# B&R Automation Studio project KeePakST401VersionX (part 5)

#### SafetySample.st
```iecst
(********************************************************************
 * COPYRIGHT -- Bernecker + Rainer
 ********************************************************************
 * Program: SafetySample
 * File: SafetySample.st
 * Author: B&R
 ********************************************************************
 * Implementation of program SafetySample
 ********************************************************************)

PROGRAM _INIT

(*KEEPAK specific hard coded values *)
	remotecmd.Password 			:= 'safety';				(* password *)
	remotecmd.NewPassword	 	:= 'safety';				(* password *)
	appcmd1.Password 			:= 'safety';
	datacmd1.Password 			:= 'safety';
	datacmd2.Password 			:= 'safety';

	visuUsedSLIDRemote			:= 1;
	visuUsedSLIDData			:= 1;

	slxused						:= 1;
	Station						:= 'IF6.ST4';
	visuEnableMachineOptions	:= 1;
	visuEnableModuleFlags		:= 1;

	visuLockSDP					:= 2;

(* command structure for remote control FUB *)
remotecmd.Version := safeVERSION_R107;	(* version *)
//remotecmd.Password := '';				(* password *)

(* command structure for application download *)
appcmd1.Version := safeVERSION_R107;	(* version *)
//appcmd1.Password := '';					(* password *)
appcmd1.ApplicationID := 1;				(* application id *)

(* command structure for machine options download *)
datacmd1.Version := safeVERSION_R107;								(* version *)
//datacmd1.Password := '';											(* password *)
datacmd1.pDeviceListInput := ADR(visuDeviceListInput);				(* device list *)
datacmd1.pMachineOptionsInput := ADR(dataMachineOptionsBitInput);	(* bit machine options *)
datacmd1.pModuleFlagsInput := ADR(dataModuleFlagsInput);			(* module flags *)
datacmd1.pAcknMachineOptions := ADR(dataAcknMachineOptions);		(* acknowledge information *)

(* command structure for extended machine options *)
datacmd2.Version := safeVERSION_R107;					(* version *)
//datacmd2.Password := '';								(* password *)
datacmd2.pIntDataInput := ADR(visuIntInput);			(* INT channels *)
datacmd2.NumberIntInput := 1;							(* number of INT channels *)
datacmd2.pUintDataInput := ADR(visuUintInput);			(* UINT channels *)
datacmd2.NumberUintInput := 1;							(* number of UINT channels *)
datacmd2.pDintDataInput := ADR(visuDintInput);			(* DINT channels *)
datacmd2.NumberDintInput := 1;							(* number of DINT channels *)
datacmd2.pUdintDataInput := ADR(visuUdintInput);		(* UDINT channels *)
datacmd2.NumberUdintInput := 1;							(* number of UDINT channels *)
datacmd2.pAcknMachineOptions := ADR(visuAcknExtData);	(* acknowledge information *)

(* hide elements in visualization *)
FOR xcnt := 0 TO SIZEOF(statusButtonActiv) - 1 DO
	statusButtonActiv[xcnt] := 1;
END_FOR

(* hide elements in visualization *)
statusButtonUnlockApp := 1;
statusButtonUnlockData := 1;
statusAcknInfoData := 1;
statusButtonUnlockExtData := 1;
statusAcknInfoExtData := 1;
statusDialog := 1;

(* set SafeLOGIC ID *)
visuUsedSLIDRemote := 1;
visuUsedSLIDData := 1;

END_PROGRAM

PROGRAM _CYCLIC
	(****************************************************************************************************************************************)
	(****************************************************************************************************************************************)
	(****************************************************************************************************************************************)
	(* show dialog to ackn command *)
	IF (dialogRemoteCmd = 1) THEN
		statusDialog := 0;
		dialogRemoteCmd := 0;
		indexButtonLeft := 0;
		indexButtonRight := 1;
		indexHeaderText := 0;
		IF (remotecmd.Data = safeCMD_SK_FORMAT) THEN
			indexMessageText := 0;
		ELSIF (remotecmd.Data = safeCMD_SK_XCHG) THEN
			indexMessageText := 1;
		ELSIF (remotecmd.Data = safeCMD_1_UDID_ACKN) THEN
			indexMessageText := 2;
		ELSIF (remotecmd.Data = safeCMD_2_UDID_ACKN) THEN
			indexMessageText := 3;
		ELSIF (remotecmd.Data = safeCMD_3_UDID_ACKN) THEN
			indexMessageText := 4;
		ELSIF (remotecmd.Data = safeCMD_4_UDID_ACKN) THEN
			indexMessageText := 5;
		ELSIF (remotecmd.Data =  safeCMD_N_UDID_ACKN) THEN
			indexMessageText := 6;
		ELSIF (remotecmd.Data =  safeCMD_CLEAR_DATA) THEN
			indexMessageText := 7;
		ELSIF (remotecmd.Data = safeCMD_FW_ACKN) THEN
			indexMessageText := 8;
		ELSIF (remotecmd.Data = safeCMD_RESET) THEN
			indexMessageText := 9;
		END_IF
	END_IF

	(* if dialog is ackn execute fub *)
	IF (dialogButtonLeft = 1 AND indexHeaderText = 0) THEN
		executeRemoteCmd := 1;
		dialogButtonLeft := 0;
		statusDialog := 1;
	ELSIF (dialogButtonRight = 1 AND indexHeaderText = 0) THEN
		dialogButtonRight := 0;
		statusDialog := 1;
	END_IF

	(* password must be at least 6 characters long *)
	IF brsstrlen(ADR(remotecmd.NewPassword)) < 6 THEN
		statusSetPassword := 2;
	ELSE
		statusSetPassword := 0;
	END_IF

	safeRemoteControl_0(SafeLOGICID := visuUsedSLIDRemote, Execute := executeRemoteCmd, pCommandData := ADR(remotecmd));
	(* reset execution flag *)
	IF (safeRemoteControl_0.Done = 1 OR safeRemoteControl_0.Error = 1) THEN
		executeRemoteCmd := 0;
	END_IF

	(* variables for visualization *)
	IF (safeRemoteControl_0.SafeLOGICStatus.SafeKEYChanged = 1) THEN
		FOR xcnt := 0 TO SIZEOF(statusButtonActiv) - 1 DO
			statusButtonActiv[xcnt] := 1;
 			statusButtonInactiv[xcnt] := 0;
		END_FOR
		statusButtonActiv[1] := 0;
 		statusButtonInactiv[1] := 1;
	ELSIF (safeRemoteControl_0.SafeLOGICStatus.NumberOfUDIDMismatches = 1 AND safeRemoteControl_0.SafeLOGICStatus.Scanning = 0) THEN
		FOR xcnt := 0 TO SIZEOF(statusButtonActiv) - 1 DO
			statusButtonActiv[xcnt] := 1;
 			statusButtonInactiv[xcnt] := 0;
		END_FOR
		statusButtonActiv[3] := 0;
 		statusButtonInactiv[3] := 1;
	ELSIF (safeRemoteControl_0.SafeLOGICStatus.NumberOfUDIDMismatches = 2 AND safeRemoteControl_0.SafeLOGICStatus.Scanning = 0) THEN
		FOR xcnt := 0 TO SIZEOF(statusButtonActiv) - 1 DO
			statusButtonActiv[xcnt] := 1;
 			statusButtonInactiv[xcnt] := 0;
		END_FOR
		statusButtonActiv[4] := 0;
 		statusButtonInactiv[4] := 1;
	ELSIF (safeRemoteControl_0.SafeLOGICStatus.NumberOfUDIDMismatches = 3 AND safeRemoteControl_0.SafeLOGICStatus.Scanning = 0) THEN
		FOR xcnt := 0 TO SIZEOF(statusButtonActiv) - 1 DO
			statusButtonActiv[xcnt] := 1;
 			statusButtonInactiv[xcnt] := 0;
		END_FOR
		statusButtonActiv[5] := 0;
 		statusButtonInactiv[5] := 1;
	ELSIF (safeRemoteControl_0.SafeLOGICStatus.NumberOfUDIDMismatches = 4 AND safeRemoteControl_0.SafeLOGICStatus.Scanning = 0) THEN
		FOR xcnt := 0 TO SIZEOF(statusButtonActiv) - 1 DO
			statusButtonActiv[xcnt] := 1;
 			statusButtonInactiv[xcnt] := 0;
		END_FOR
		statusButtonActiv[6] := 0;
 		statusButtonInactiv[6] := 1;
	ELSIF (safeRemoteControl_0.SafeLOGICStatus.NumberOfUDIDMismatches > 4 AND safeRemoteControl_0.SafeLOGICStatus.Scanning = 0) THEN
		FOR xcnt := 0 TO SIZEOF(statusButtonActiv) - 1 DO
			statusButtonActiv[xcnt] := 1;
 			statusButtonInactiv[xcnt] := 0;
		END_FOR
		statusButtonActiv[7] := 0;
 		statusButtonInactiv[7] := 1;
	ELSIF (safeRemoteControl_0.SafeLOGICStatus.NumberOfDifferentFirmware <> 0 AND safeRemoteControl_0.SafeLOGICStatus.Scanning = 0) THEN
		FOR xcnt := 0 TO SIZEOF(statusButtonActiv) - 1 DO
			statusButtonActiv[xcnt] := 1;
 			statusButtonInactiv[xcnt] := 0;
		END_FOR
		statusButtonActiv[11] := 0;
 		statusButtonInactiv[11] := 1;
	ELSE
		FOR xcnt := 0 TO SIZEOF(statusButtonActiv) - 1 DO
			statusButtonActiv[xcnt] := 1;
 			statusButtonInactiv[xcnt] := 0;
		END_FOR
	END_IF
	(* status text - MXCHG *)
	IF (safeRemoteControl_0.SafeLOGICStatus.LedTestActive = 1) THEN
		indexMxchgLed := 40;
	ELSIF (safeRemoteControl_0.SafeLOGICStatus.Scanning = 1) THEN
		indexMxchgLed := 30;
	ELSIF (safeRemoteControl_0.SafeLOGICStatus.NumberOfUDIDMismatches = 1) THEN
		indexMxchgLed := 1;
	ELSIF (safeRemoteControl_0.SafeLOGICStatus.NumberOfUDIDMismatches = 2) THEN
		indexMxchgLed := 2;
	ELSIF (safeRemoteControl_0.SafeLOGICStatus.NumberOfUDIDMismatches = 3) THEN
		indexMxchgLed := 3;
	ELSIF (safeRemoteControl_0.SafeLOGICStatus.NumberOfUDIDMismatches = 4) THEN
		indexMxchgLed := 4;
	ELSIF (safeRemoteControl_0.SafeLOGICStatus.NumberOfUDIDMismatches > 4) THEN
		indexMxchgLed := 5;
	ELSIF (safeRemoteControl_0.SafeLOGICStatus.NumberOfMissingModules <> 0) THEN
		indexMxchgLed := 20;
	ELSIF (safeRemoteControl_0.SafeLOGICStatus.NumberOfUDIDMismatches = 0) THEN
		indexMxchgLed := 10;
	END_IF
	(* status text - FW-ACKN *)
	IF (safeRemoteControl_0.SafeLOGICStatus.SafeKEYChanged = 0 AND safeRemoteControl_0.SafeLOGICStatus.NumberOfDifferentFirmware = 0) THEN
		indexFwAcknLed := 10;
	ELSIF (safeRemoteControl_0.SafeLOGICStatus.SafeKEYChanged = 1) THEN
		indexFwAcknLed := 1;
	ELSIF (safeRemoteControl_0.SafeLOGICStatus.NumberOfDifferentFirmware <> 0) THEN
		indexFwAcknLed := 2;
	END_IF
	(* status text - FAIL *)
	IF (safeRemoteControl_0.SafeLOGICStatus.FailSafe <> 16#55) THEN
		indexFAILLed := 2;
	ELSIF (safeRemoteControl_0.SafeLOGICStatus.openSAFETYstate = 0) THEN
		indexFAILLed := 0;
	ELSIF (safeRemoteControl_0.SafeLOGICStatus.openSAFETYstate = 1) THEN
		indexFAILLed := 1;
	END_IF
	(* status text - R/E *)
	indexRELed := safeRemoteControl_0.SafeLOGICStatus.SafeOSState;

	(****************************************************************************************************************************************)
	(****************************************************************************************************************************************)
	(****************************************************************************************************************************************)
	(* show dialog to ackn command *)
	IF (dialogApplication = 1) THEN
		statusDialog := 0;
		dialogApplication := 0;
		indexButtonLeft := 0;
		indexButtonRight := 1;
		indexHeaderText := 1;
		indexMessageText := 10;
	END_IF

	(* if dialog is ackn unlock application *)
	IF (dialogButtonLeft = 1 AND indexHeaderText = 1) THEN
		appcmd1.Unlock := 1;
		dialogButtonLeft := 0;
		statusDialog := 1;
	ELSIF (dialogButtonRight = 1 AND indexHeaderText = 1) THEN
		appcmd1.Unlock := 2;
		dialogButtonRight := 0;
		statusDialog := 1;
	END_IF

	(* convert application CRC to HEX string *)
	itoahex(safeDownloadApplication_0.ApplicationCRC, ADR(visuApplicationCRC));

	safeDownloadApplication_0(SafeLOGICID := appcmd1.ApplicationID, Execute := executeapp1, pCommandData := ADR(appcmd1));

	(* show unlock button *)
	IF (safeDownloadApplication_0.UnlockRequired = 1) THEN
		statusButtonUnlockApp := 0;
	ELSE
		appcmd1.Unlock := 0;
		statusButtonUnlockApp := 1;
	END_IF

	(****************************************************************************************************************************************)
	(****************************************************************************************************************************************)
	(****************************************************************************************************************************************)
	(* disable machine options *)
	IF (visuEnableMachineOptions = FALSE) THEN
		datacmd1.pMachineOptionsInput := 0;
	ELSE
		datacmd1.pMachineOptionsInput := ADR(dataMachineOptionsBitInput);
	END_IF

	(* disable module flags *)
	IF (visuEnableModuleFlags = FALSE) THEN
		datacmd1.pModuleFlagsInput := 0;
	ELSE
		datacmd1.pModuleFlagsInput := ADR(dataModuleFlagsInput);
	END_IF

	(* Machine Option Bit #000 *)
	IF (visuMachineOptionsBitInput[0] = 1) THEN
		dataMachineOptionsBitInput.BitData[0].0 := 1;
	ELSE
		dataMachineOptionsBitInput.BitData[0].0 := 0;
	END_IF
	(* Machine Option Bit #001 *)
	IF (visuMachineOptionsBitInput[1] = 1) THEN
		dataMachineOptionsBitInput.BitData[0].1 := 1;
	ELSE
		dataMachineOptionsBitInput.BitData[0].1 := 0;
	END_IF
	(* Machine Option Bit #002 *)
	IF (visuMachineOptionsBitInput[2] = 1) THEN
		dataMachineOptionsBitInput.BitData[0].2 := 1;
	ELSE
		dataMachineOptionsBitInput.BitData[0].2 := 0;
	END_IF
	(* Optional Flag Module #1 *)
	IF (visuModuleFlagsOptionalInput[1] = 1) THEN
		dataModuleFlagsInput.Optional[0].1 := 1;
	ELSE
		dataModuleFlagsInput.Optional[0].1 := 0;
	END_IF
	(* Optional Flag Module #2 *)
	IF (visuModuleFlagsOptionalInput[2] = 1) THEN
		dataModuleFlagsInput.Optional[0].2 := 1;
	ELSE
		dataModuleFlagsInput.Optional[0].2 := 0;
	END_IF
	(* Startup Flag Module #1 *)
	IF (visuModuleFlagsStartupInput[1] = 1) THEN
		dataModuleFlagsInput.Startup[0].1 := 1;
	ELSE
		dataModuleFlagsInput.Startup[0].1 := 0;
	END_IF
	(* Startup Flag Module #2 *)
	IF (visuModuleFlagsStartupInput[2] = 1) THEN
		dataModuleFlagsInput.Startup[0].2 := 1;
	ELSE
		dataModuleFlagsInput.Startup[0].2 := 0;
	END_IF
	(* Not_Present Flag Module #1 *)
	IF (visuModuleFlagsNotPresentInput[1] = 1) THEN
		dataModuleFlagsInput.NotPresent[0].1 := 1;
	ELSE
		dataModuleFlagsInput.NotPresent[0].1 := 0;
	END_IF
	(* Not_Present Flag Module #2 *)
	IF (visuModuleFlagsNotPresentInput[2] = 1) THEN
		dataModuleFlagsInput.NotPresent[0].2 := 1;
	ELSE
		dataModuleFlagsInput.NotPresent[0].2 := 0;
	END_IF

	(* Ackn Machine Option Bit #000 *)
	IF (visuAcknMachineOptions[0] = 1) THEN
		dataAcknMachineOptions.AcknBitOptions[0].0 := 1;
	ELSE
		dataAcknMachineOptions.AcknBitOptions[0].0 := 0;
	END_IF
	(* Ackn Machine Option Bit #001 *)
	IF (visuAcknMachineOptions[1] = 1) THEN
		dataAcknMachineOptions.AcknBitOptions[0].1 := 1;
	ELSE
		dataAcknMachineOptions.AcknBitOptions[0].1 := 0;
	END_IF
	(* Ackn Machine Option Bit #002 *)
	IF (visuAcknMachineOptions[2] = 1) THEN
		dataAcknMachineOptions.AcknBitOptions[0].2 := 1;
	ELSE
		dataAcknMachineOptions.AcknBitOptions[0].2 := 0;
	END_IF

	(* show dialog to ackn command *)
	IF (dialogData = 1) THEN
		statusDialog := 0;
		dialogData := 0;
		indexButtonLeft := 0;
		indexButtonRight := 1;
		indexHeaderText := 2;
		indexMessageText := 11;
	END_IF

	(* if dialog is ackn unlock data *)
	IF (dialogButtonLeft = 1 AND indexHeaderText = 2) THEN
		datacmd1.Unlock := 1;
		dialogButtonLeft := 0;
		statusDialog := 1;
	ELSIF (dialogButtonRight = 1 AND indexHeaderText = 2) THEN
		datacmd1.Unlock := 2;
		dialogButtonRight := 0;
		statusDialog := 1;
	END_IF

	safeDownloadData_0(SafeLOGICID := visuUsedSLIDData, Execute := executedata1, Type:= safeDATA_TYPE_MAOP, pCommandData := ADR(datacmd1));

	(* data compare failed *)
	IF (safeDownloadData_0.StatusID = safeERR_DL_COMPARE_FAILED) THEN
		indexCompareTextData := 2;
	ELSE
		indexCompareTextData := 0;
	END_IF

	IF (safeDownloadData_0.UnlockRequired = 1) THEN
		(* data compare successful *)
		indexCompareTextData := 1;
		IF (datacmd1.pDeviceListOutput <> 0 AND datacmd1.NumberDevicesOutput <> 0) THEN
			pDeviceListOut ACCESS datacmd1.pDeviceListOutput;

			(* device #1 *)
			visuDeviceListOutput[0].SADR := pDeviceListOut[0].SADR;
			brsmemcpy(ADR(visuDeviceListOutput[0].UDID_High), ADR(pDeviceListOut[0].UDID[0]), 2);
			(* swap UDID *)
			visuDeviceListOutput[0].UDID_High := swapUINT(visuDeviceListOutput[0].UDID_High);
			brsmemcpy(ADR(visuDeviceListOutput[0].UDID_Low), ADR(pDeviceListOut[0].UDID[2]), 4);
			(* swap UDID *)
			visuDeviceListOutput[0].UDID_Low := swapUDINT(visuDeviceListOutput[0].UDID_Low);
			(* device #2 *)
			visuDeviceListOutput[1].SADR := pDeviceListOut[1].SADR;
			brsmemcpy(ADR(visuDeviceListOutput[1].UDID_High), ADR(pDeviceListOut[1].UDID[0]), 2);
			(* swap UDID *)
			visuDeviceListOutput[1].UDID_High := swapUINT(visuDeviceListOutput[1].UDID_High);
			brsmemcpy(ADR(visuDeviceListOutput[1].UDID_Low), ADR(pDeviceListOut[1].UDID[2]), 4);
			(* swap UDID *)
			visuDeviceListOutput[1].UDID_Low := swapUDINT(visuDeviceListOutput[1].UDID_Low);
		END_IF

		IF (datacmd1.pMachineOptionsOutput <> 0) THEN
			pMachineOptionsBitOut ACCESS datacmd1.pMachineOptionsOutput;

			(* Machine Option Bit #000 *)
			IF (pMachineOptionsBitOut.BitData[0].0 = 1) THEN
				visuMachineOptionsBitOutput[0] := 1;
			END_IF
			(* Machine Option Bit #001 *)
			IF (pMachineOptionsBitOut.BitData[0].1 = 1) THEN
				visuMachineOptionsBitOutput[1] := 1;
			END_IF
			(* Machine Option Bit #002 *)
			IF (pMachineOptionsBitOut.BitData[0].2 = 1) THEN
				visuMachineOptionsBitOutput[2] := 1;
			END_IF
		END_IF

		IF (datacmd1.pModuleFlagsOutput <> 0) THEN
			pModuleFlagsOut ACCESS datacmd1.pModuleFlagsOutput;

			(* Optional Flag Module #1 *)
			IF (pModuleFlagsOut.Optional[0].1 = 1) THEN
				visuModuleFlagsOptionalOutput[1] := 1;
			END_IF
			(* Optional Flag Module #2 *)
			IF (pModuleFlagsOut.Optional[0].2 = 1) THEN
				visuModuleFlagsOptionalOutput[2] := 1;
			END_IF
			(* Startup Flag Module #1 *)
			IF (pModuleFlagsOut.Startup[0].1 = 1) THEN
				visuModuleFlagsStartupOutput[1] := 1;
			END_IF
			(* Startup Flag Module #2 *)
			IF (pModuleFlagsOut.Startup[0].2 = 1) THEN
				visuModuleFlagsStartupOutput[2] := 1;
			END_IF
			(* Not_Present Flag Module #1 *)
			IF (pModuleFlagsOut.NotPresent[0].1 = 1) THEN
				visuModuleFlagsNotPresentOutput[1] := 1;
			END_IF
			(* Not_Present Flag Module #2 *)
			IF (pModuleFlagsOut.NotPresent[0].2 = 1) THEN
				visuModuleFlagsNotPresentOutput[2] := 1;
			END_IF
		END_IF
		(* show ackn box *)
		statusAcknInfoData := 0;
		(* show unlock button unlocked if one ACK is set *)
		IF (visuAcknMachineOptions[0] = 1 OR visuAcknMachineOptions[1] = 1 OR visuAcknMachineOptions[2] = 1) THEN
			statusButtonUnlockData := 0;
		END_IF
	ELSIF (safeDownloadData_0.Done = 1 OR safeDownloadData_0.Error = 1) THEN
		(* reset visualization elements *)
		brsmemset(ADR(visuDeviceListOutput), 0, SIZEOF(visuDeviceListOutput));
		brsmemset(ADR(visuMachineOptionsBitOutput), 0, SIZEOF(visuMachineOptionsBitOutput));
		brsmemset(ADR(visuModuleFlagsOptionalOutput), 0, SIZEOF(visuModuleFlagsOptionalOutput));
		brsmemset(ADR(visuModuleFlagsStartupOutput), 0, SIZEOF(visuModuleFlagsStartupOutput));
		brsmemset(ADR(visuModuleFlagsNotPresentOutput), 0, SIZEOF(visuModuleFlagsNotPresentOutput));
		(* hide ackn box *)
		statusAcknInfoData := 1;
		(* hide unlock button *)
		datacmd1.Unlock := 0;
		statusButtonUnlockData := 1;
		(* reset ackn flags *)
		visuAcknMachineOptions[0] := 0;
		visuAcknMachineOptions[1] := 0;
		visuAcknMachineOptions[2] := 0;
	ELSE
		(* hide ackn box *)
		statusAcknInfoData := 1;
		(* hide unlock button *)
		datacmd1.Unlock := 0;
		statusButtonUnlockData := 1;
	END_IF

	(****************************************************************************************************************************************)
	(****************************************************************************************************************************************)
	(****************************************************************************************************************************************)
	(* Enable for INT set *)
	IF (visuEnableINTOptions <> 0) THEN
		datacmd2.pIntDataInput := ADR(visuIntInput);
		datacmd2.NumberIntInput := 1;
	ELSE
		datacmd2.pIntDataInput := 0;
		datacmd2.NumberIntInput := 0;
	END_IF
	(* Enable for UINT set *)
	IF (visuEnableUINTOptions <> 0) THEN
		datacmd2.pUintDataInput := ADR(visuUintInput);
		datacmd2.NumberUintInput := 1;
	ELSE
		datacmd2.pUintDataInput := 0;
		datacmd2.NumberUintInput := 0;
	END_IF
	(* Enable for DINT set *)
	IF (visuEnableDINTOptions <> 0) THEN
		datacmd2.pDintDataInput := ADR(visuDintInput);
		datacmd2.NumberDintInput := 1;
	ELSE
		datacmd2.pDintDataInput := 0;
		datacmd2.NumberDintInput := 0;
	END_IF
	(* Enable for UDINT set *)
	IF (visuEnableUDINTOptions <> 0) THEN
		datacmd2.pUdintDataInput := ADR(visuUdintInput);
		datacmd2.NumberUdintInput := 1;
	ELSE
		datacmd2.pUdintDataInput := 0;
		datacmd2.NumberUdintInput := 0;
	END_IF

	(* show dialog to ackn command *)
	IF (dialogExtData = 1) THEN
		statusDialog := 0;
		dialogExtData := 0;
		indexButtonLeft := 0;
		indexButtonRight := 1;
		indexHeaderText := 3;
		indexMessageText := 11;
	END_IF

	(* if dialog is ackn unlock data *)
	IF (dialogButtonLeft = 1 AND indexHeaderText = 3) THEN
		datacmd2.Unlock := 1;
		dialogButtonLeft := 0;
		statusDialog := 1;
	ELSIF (dialogButtonRight = 1 AND indexHeaderText = 3) THEN
		datacmd2.Unlock := 2;
		dialogButtonRight := 0;
		statusDialog := 1;
	END_IF

	safeDownloadData_1(SafeLOGICID := visuUsedSLIDData, Execute := executedata2, Type:= safeDATA_TYPE_EXTMAOP, pCommandData := ADR(datacmd2));

	(* data compare failed *)
	IF (safeDownloadData_1.StatusID = safeERR_DL_COMPARE_FAILED) THEN
		indexCompareTextExtData := 2;
	ELSE
		indexCompareTextExtData := 0;
	END_IF

	IF (safeDownloadData_1.UnlockRequired = 1) THEN
		(* data compare successful *)
		indexCompareTextExtData := 1;

		(* INT channels *)
		IF (datacmd2.pIntDataOutput <> 0 AND datacmd2.NumberIntOutput <> 0) THEN
			brsmemcpy(ADR(visuIntOutput), datacmd2.pIntDataOutput, SIZEOF(visuIntOutput));
		END_IF
		(* UINT channels *)
		IF (datacmd2.pUintDataOutput <> 0 AND datacmd2.NumberUintOutput <> 0) THEN
			brsmemcpy(ADR(visuUintOutput), datacmd2.pUintDataOutput, SIZEOF(visuUintOutput));
		END_IF
		(* DINT channels *)
		IF (datacmd2.pDintDataOutput <> 0 AND datacmd2.NumberDintOutput <> 0) THEN
			brsmemcpy(ADR(visuDintOutput), datacmd2.pDintDataOutput, SIZEOF(visuDintOutput));
		END_IF
		(* UDINT channels *)
		IF (datacmd2.pUdintDataOutput <> 0 AND datacmd2.NumberUdintOutput <> 0) THEN
			brsmemcpy(ADR(visuUdintOutput), datacmd2.pUdintDataOutput, SIZEOF(visuUdintOutput));
		END_IF
		(* show ackn box *)
		statusAcknInfoExtData := 0;
		(* show unlock button if one ACK is set *)
		IF (visuAcknExtData.AcknIntOptions[0] = 1 OR visuAcknExtData.AcknUintOptions[0] = 1 OR visuAcknExtData.AcknDintOptions[0] = 1 OR visuAcknExtData.AcknUdintOptions[0] = 1) THEN
			statusButtonUnlockExtData := 0;
		END_IF
	ELSIF (safeDownloadData_1.Done = 1 OR safeDownloadData_1.Error = 1) THEN
		(* reset visualization elements *)
		brsmemset(ADR(visuIntOutput), 0, SIZEOF(visuIntOutput));
		brsmemset(ADR(visuUintOutput), 0, SIZEOF(visuUintOutput));
		brsmemset(ADR(visuDintOutput), 0, SIZEOF(visuDintOutput));
		brsmemset(ADR(visuUdintOutput), 0, SIZEOF(visuUdintOutput));
		(* hide ackn box *)
		statusAcknInfoExtData := 1;
		(* hide unlock button *)
		datacmd2.Unlock := 0;
		statusButtonUnlockExtData := 1;
		(* reset ackn flags *)
		visuAcknExtData.AcknIntOptions[0] := 0;
		visuAcknExtData.AcknUintOptions[0] := 0;
		visuAcknExtData.AcknDintOptions[0] := 0;
		visuAcknExtData.AcknUdintOptions[0] := 0;
	ELSE
		(* hide ackn box *)
		statusAcknInfoExtData := 1;
		(* hide unlock button *)
		datacmd2.Unlock := 0;
		statusButtonUnlockExtData := 1;
	END_IF

	(****************************************************************************************************************************************)
	(****************************************************************************************************************************************)
	(****************************************************************************************************************************************)
	(* read UDID from SafeLOGIC-X *)
	IF slxused = 1 THEN
		readUDIDlowSLX(enable := 1, pDeviceName := ADR(Station), pChannelName := ADR('UDID_low'));

		IF readUDIDlowSLX.status = 0 THEN
			UDID_Low := readUDIDlowSLX.value;
		ELSIF readUDIDlowSLX.status <> 65535 THEN
			UDID_Low := 0;
		END_IF

		readUDIDhighSLX(enable := 1, pDeviceName := ADR(Station), pChannelName := ADR('UDID_high'));

		IF readUDIDhighSLX.status = 0 THEN
			UDID_High := UDINT_TO_UINT(readUDIDhighSLX.value);
		ELSIF readUDIDhighSLX.status <> 65535 THEN
			UDID_High := 0;
		END_IF

		(* hide / show visualization elements *)
		stautsSLXInformation := 0;
		statusSLInformation := 1;
	(* read UDID form SafeLOGIC *)
	ELSE
		readUDIDlowSL(enable := 1, pDevice := ADR(Interface), node := Node, index := 16#2000, subindex := 6, pData := ADR(UDID_Low), datalen := SIZEOF(UDID_Low));

		IF readUDIDlowSL.status <> 0 AND readUDIDlowSL.status <> 65535 THEN
			UDID_Low := 0;
		END_IF

		readUDIDhighSL(enable := 1, pDevice := ADR(Interface), node := Node, index := 16#2000, subindex := 7, pData := ADR(UDID_High), datalen := SIZEOF(UDID_High));

		IF readUDIDhighSL.status <> 0 AND readUDIDhighSL.status <> 65535 THEN
			UDID_High := 0;
		END_IF

		(* hide / show visualization elements *)
		stautsSLXInformation := 1;
		statusSLInformation := 0;
	END_IF

	(* convert UDID to HEX string *)
	itoahex(UDID_Low, ADR(visuUDID_Low));
	itoahex(UDID_High, ADR(visuUDID_High));

	(****************************************************************************************************************************************)
	(****************************************************************************************************************************************)
	(****************************************************************************************************************************************)
	(* write UDID for SafeLOGIC to command structure *)
	appcmd1.UDID_Low := UDID_Low;
	appcmd1.UDID_High := UDID_High;
	datacmd1.UDID_Low := UDID_Low;
	datacmd1.UDID_High := UDID_High;
	datacmd2.UDID_Low := UDID_Low;
	datacmd2.UDID_High := UDID_High;

END_PROGRAM
```

### Package Logical/ServoMotion - gServoRamobj

### Program Logical/ServoMotion/ServoRamHandler (IEC)

#### Main.st - Init, cyclic, exit code
```iecst
PROGRAM _INIT
	(* Insert code here *)

    gHMI.Parameters.ServoRamJogVelocity := 50;
    gHMI.Parameters.ServoRamPositiveVelocity := 650.0;
    gHMI.Parameters.ServoRamNegativeVelocity := 950.0;
    gHMI.Parameters.ServoRamAccel := 5000.0;

    gHMI.Parameters.ServoRamStartPosition := 50.0;
    gHMI.Parameters.ServoRamEndPosition := 500.0;

    gHMI.Parameters.ServoRamEndDwellTime := 2000;
    gHMI.Parameters.ServoRamStartDwellTime := 100;

    gHMI.Parameters.ServoRamTorqueLimit := 6.0;
    gHMI.Parameters.ServoRamClearPosition := 300;

    gPassword; //need to use this somewhere. Was getting thrown out in slimmed down test code for servo ram

    TON_RamDelay(IN := gIO.DIs.BodyDetect , PT := RamDelay );

END_PROGRAM

PROGRAM _CYCLIC

    IF gHighSeverityAlarmActive THEN
        state := SERVORAM_ERROR;
    END_IF

    gIO.DOs.ResetSafety := gHMI.Commands.RequestReset;

    StartDwellTimer.IN := FALSE; //Set in state machine if needed
    EndDwellTimer.IN := FALSE;

    IF gServoRamInterface.Status.ActualPosition <= gHMI.Parameters.ServoRamClearPosition THEN
        ServoRamClear := TRUE;
    ELSE
        ServoRamClear := FALSE;
    END_IF

    IF NOT gHMI.Commands.CycleServoRam THEN
        state := SERVORAM_IDLE;
    END_IF

    CASE state OF

        SERVORAM_WAIT_FOR_HOME:

            //servo ram should home automatically on machine start up.
            IF gServoRamInterface.Status.Homed AND ServoRamFirstHomeExecuted THEN
                ServoRamAutoHome := FALSE;
                gRamAtStopPosition := TRUE;
                gHMI.Commands.CycleServoRam := FALSE;
                gServoRamInterface.Commands.ToMapp.TorqueLimitingOn := TRUE; //turn torque limiting on
                state := SERVORAM_IDLE;
            ELSIF gServoRamInterface.Status.PoweredOn THEN
                ServoRamAutoHome := TRUE;
            END_IF

        SERVORAM_IDLE:

            IF gHMI.Commands.CycleServoRam AND ServoRamFirstHomeExecuted THEN
                ServoRamBusy := TRUE;
                gServoRamInterface.Commands.ToMapp.TorqueLimitingOn := TRUE; //turn torque limiting on

                gServoRamInterface.Parameters.MovementParameters.Position := gHMI.Parameters.ServoRamStartPosition;
                gServoRamInterface.Parameters.MovementParameters.Velocity := gHMI.Parameters.ServoRamPositiveVelocity;
                gServoRamInterface.Commands.RequestMoveAbs := TRUE;

                state := SERVORAM_MOVE_TO_START;
            END_IF

        SERVORAM_WAITING_ON_BOX:

            IF (gIO.DIs.BodyDetect AND (gModeControlInterface.Commands.SetShowMode = FALSE)) OR
                (gIO.DIs.X_BlowOff AND gModeControlInterface.Commands.SetShowMode) THEN

                FeedInCycle := FALSE;

                gServoRamInterface.Parameters.MovementParameters.Position := gHMI.Parameters.ServoRamEndPosition;
                gServoRamInterface.Parameters.MovementParameters.Velocity := gHMI.Parameters.ServoRamPositiveVelocity;
                gRamAtStopPosition := FALSE;
                gServoRamInterface.Commands.RequestMoveAbs := TRUE;
                ServoRamBusy := TRUE ;

                state := SERVORAM_MOVE_TO_END;
            END_IF

        SERVORAM_MOVE_TO_END:

            gIO.DOs.PushOn := gPusherOn;

            IF gServoRamInterface.Status.MoveComplete THEN
                gServoRamInterface.Status.MoveComplete := FALSE;

                gServoRamInterface.Commands.ToMapp.Update := TRUE; //This forces update of the torque limit. This will be cleared automatically

                IF gHMI.Parameters.ServoRamEndDwellTime > 0 THEN

                    EndDwellTimer.IN := TRUE;
                    state := SERVORAM_DWELL_AT_END;
                ELSE

                    CycleCount := CycleCount + 1;
                    LubeCount := LubeCount + 1;

                    gServoRamInterface.Parameters.MovementParameters.Position := gHMI.Parameters.ServoRamStartPosition;
                    gServoRamInterface.Parameters.MovementParameters.Velocity := gHMI.Parameters.ServoRamNegativeVelocity;
                    gServoRamInterface.Commands.RequestMoveAbs := TRUE;

                    state := SERVORAM_MOVE_TO_START;

                END_IF
            END_IF

        SERVORAM_DWELL_AT_END:

            EndDwellTimer.IN := TRUE;

            IF EndDwellTimer.Q THEN
                EndDwellTimer.IN := FALSE;

                CycleCount := CycleCount + 1;

                gServoRamInterface.Parameters.MovementParameters.Position := gHMI.Parameters.ServoRamStartPosition;
                gServoRamInterface.Parameters.MovementParameters.Velocity := gHMI.Parameters.ServoRamNegativeVelocity;
                gServoRamInterface.Commands.RequestMoveAbs := TRUE;

                state := SERVORAM_MOVE_TO_START;

            END_IF

        SERVORAM_MOVE_TO_START:

            IF gServoRamInterface.Status.MoveComplete THEN
                gRamAtStopPosition := TRUE;
                gServoRamInterface.Status.MoveComplete := FALSE;
                ServoRamBusy := FALSE;

                IF NOT(FeedInCycle) THEN
                    gModeControlInterface.Commands.FinishCycle := FALSE;
                END_IF

                IF gHMI.Parameters.ServoRamStartDwellTime > 0 THEN

                    EndDwellTimer.IN := TRUE;
                    state := SERVORAM_DWELL_AT_START;
                ELSE

                    state := SERVORAM_WAITING_ON_BOX;
                END_IF

            END_IF

        SERVORAM_DWELL_AT_START:

            StartDwellTimer.IN := TRUE;

            IF StartDwellTimer.Q THEN
                StartDwellTimer.IN := FALSE;

                state := SERVORAM_IDLE;
            END_IF

        SERVORAM_ERROR:

            ServoRamAutoHome := FALSE;
            gServoRamInterface.Status.MoveComplete := FALSE;
            gHMI.Commands.CycleServoRam := FALSE;
            ServoRamBusy := FALSE;
            ServoRamAutoHome := FALSE;

            IF (gNumActiveAlarms = 0) THEN
                state := SERVORAM_WAIT_FOR_HOME;
            END_IF

    END_CASE;

    StartDwellTimer.PT := gHMI.Parameters.ServoRamStartDwellTime;
    StartDwellTimer();

    //EndDwellTimer.PT := gHMI.Parameters.ServoRamEndDwellTime;
    EndDwellTimer.PT := gHMI.Parameters.ServoRamEndDwellTime; //Use existing dwell time from HMI
    EndDwellTimer();

				END_PROGRAM

PROGRAM _EXIT
				(* Insert code here *)

				END_PROGRAM
```

#### Types.typ - Local data types
```iecst
TYPE
	ServoRamState_enum :
		(
		SERVORAM_WAIT_FOR_HOME := 0,
		SERVORAM_IDLE := 10,
		SERVORAM_WAITING_ON_BOX := 15,
		SERVORAM_MOVE_TO_END := 20,
		SERVORAM_DWELL_AT_END := 40,
		SERVORAM_MOVE_TO_START := 60,
		SERVORAM_DWELL_AT_START := 80,
		SERVORAM_ERROR := 999
		);
END_TYPE
```

#### Variables.var - Local variables
```iecst
VAR
	StartDwellTimer : TON;
	EndDwellTimer : TON;
	state : ServoRamState_enum;
END_VAR
```

### Program Logical/ServoMotion/ServoFeedHandler (IEC)

#### Main.st - Init, cyclic, exit code
```iecst
PROGRAM _INIT
	(* Insert code here *)

    gHMI.Parameters.ServoFeedJogVelocity := 50;
    gHMI.Parameters.ServoFeedVelocity := 600.0;
    gHMI.Parameters.ServoFeedAccel := 600.0;
    HoperLowStop;

END_PROGRAM

PROGRAM _CYCLIC

//	IF gNumActiveAlarms  > 0 THEN
//		state := SERVOFEED_ERROR;
//	END_IF

    IF gHighSeverityAlarmActive THEN
        state := SERVOFEED_ERROR;
    END_IF

    CASE state OF

        SERVOFEED_WAIT_FOR_HOME:

            //servo ram should home automatically on machine start up. This is a direct home axis and should not rquire a home command
            IF gServoFeedInterface.Status.Homed THEN
                state := SERVOFEED_IDLE;
            END_IF

        SERVOFEED_IDLE:

            IF gHMI.Commands.StartServoFeed AND ServoFeedFirstHomeExecuted THEN

                gServoFeedInterface.Commands.RequestMoveVelocity := TRUE;

                state := SERVOFEED_MOVE_VELOCITY;
            END_IF

        SERVOFEED_MOVE_VELOCITY:

            //Added gDownstreamBlocked := TRUE. 07-14-22.
            IF gHMI.Commands.StartServoFeed = FALSE OR gDownstreamBlocked = TRUE THEN
                gServoFeedInterface.Commands.RequestMoveVelocity := FALSE;

                state := SERVOFEED_IDLE;
                //                END_IF
            END_IF

        SERVOFEED_ERROR:

            gServoFeedInterface.Status.MoveComplete := FALSE;
            gHMI.Commands.StartServoFeed := FALSE;

            gServoFeedInterface.Commands.RequestMoveVelocity := FALSE;

            IF (gNumActiveAlarms = 0) THEN
                state := SERVOFEED_WAIT_FOR_HOME;
            END_IF

    END_CASE;
	FeedStopTimer();
END_PROGRAM

PROGRAM _EXIT
				(* Insert code here *)

END_PROGRAM
```

#### Types.typ - Local data types
```iecst
TYPE
	ServoFeedState_enum :
		(
		SERVOFEED_WAIT_FOR_HOME := 0,
		SERVOFEED_IDLE := 10,
		SERVOFEED_MOVE_VELOCITY := 20,
		SERVOFEED_ERROR := 999
		);
END_TYPE
```

#### Variables.var - Local variables
```iecst
VAR
	HopperLowStop : BOOL;
	state : ServoFeedState_enum;
	FeedStopTimer : TON;
END_VAR
VAR RETAIN
	CycleCount : UDINT;
END_VAR
```

### Program Logical/ServoMotion/ServoHopperHandler (IEC)

#### Types.typ
```iecst
TYPE
	ServoHopperState_enum :
		(
		SERVOHOPPER_WAIT_FOR_HOME := 0,
		SERVOHOPPER_IDLE := 5,
		SERVOHOPPER_MOVE_VELOCITY := 10,
		SERVOHOPPER_COOLDOWN := 15,
		SERVOHOPPER_ERROR := 999,
		SERVOHOPPER_MOVE_TO_END := 20,
		SERVOHOPPER_DWELL_AT_END := 40,
		SERVOHOPPER_MOVE_TO_START := 60,
		SERVOHOPPER_DWELL_AT_START := 80
		);
END_TYPE
```

#### Variables.var
```iecst
VAR
	ResetTimeoutAlarm : BOOL;
	StartDwellTimer : TON;
	AtTorqueTimer : TON;
	state : ServoHopperState_enum;
END_VAR
VAR RETAIN
	CycleCount : UDINT;
END_VAR
VAR
	ResetTimeoutTimer : TON;
END_VAR
```

#### Main.st
```iecst
PROGRAM _INIT
	(* Insert code here *)

	gHMI.Parameters.ServoHopperJogVelocity := 3.35;
	gHMI.Parameters.ServoHopperVelocity := 3.35;
	gHMI.Parameters.ServoHopperAccel := 180.0;

	gHMI.Parameters.ServoHopperTorqueLimit := 2.5;

	gHMI.Parameters.ServoHopperDwellTime := 1500; //1 s
	gHMI.Parameters.AtTorqueTime := 500; //1 s

END_PROGRAM

PROGRAM _CYCLIC

	IF gNumActiveAlarms  > 0 THEN
		state := SERVOHOPPER_ERROR;
	END_IF

	IF gHighSeverityAlarmActive THEN
		state := SERVOHOPPER_ERROR;
	END_IF

	//make sure that torque limiting is turned on while jogging
	//	IF EDGEPOS(gHMI.Commands.JogServoHopperPos) THEN
	//		gServoHopperInterface.Commands.ToMapp.TorqueLimitingOn := TRUE;
	//	END_IF
	//	IF EDGEPOS(gHMI.Commands.JogServoHopperNeg) THEN
	//		gServoHopperInterface.Commands.ToMapp.TorqueLimitingOn := TRUE;
	//	END_IF

	StartDwellTimer.IN := FALSE; //clear otuside state machine. will  e set true in appropriate state
    AtTorqueTimer.IN := FALSE;
    ResetTimeoutTimer.IN := FALSE;

    // If the hopper has been reset but the machine isn't running, only let the hopper run for an alotted time to protect the motor
    IF gIO.DIs.HopperMotor_RUN AND (NOT gHMI.Commands.RequestVFDRun) THEN
        ResetTimeoutTimer.IN := TRUE;
    END_IF
    IF ResetTimeoutTimer.Q THEN
        ResetTimeoutAlarm := TRUE;
    END_IF

    // Resetting clears the timeout alarms
    IF gHMI.Commands.RequestReset THEN
        ResetTimeoutAlarm := FALSE;
    END_IF

	CASE state OF

		SERVOHOPPER_WAIT_FOR_HOME:

			//servo ram should home automatically on machine start up. This is a direct home axis and should not rquire a home command
			IF gServoFeedInterface.Status.Homed THEN
				gServoHopperInterface.Commands.ToMapp.TorqueLimitingOn := TRUE;
				state := SERVOHOPPER_IDLE;
			END_IF

		SERVOHOPPER_IDLE:

			IF gIO.DIs.HopperMotor_RUN AND ServoHopperFirstHomeExecuted THEN
				gServoHopperInterface.Commands.ToMapp.TorqueLimitingOn := TRUE; //turn torque limiting on

				gServoHopperInterface.Commands.RequestMoveVelocity := TRUE;
				gServoHopperInterface.Parameters.MovementParameters.Direction := 0;

				state := SERVOHOPPER_MOVE_VELOCITY;
			END_IF

		SERVOHOPPER_MOVE_VELOCITY:

			AtTorqueTimer.IN := (gServoHopperInterface.Status.ActualTorque >= gHMI.Parameters.ServoHopperTorqueLimit *0.90);

			IF gIO.DIs.HopperMotor_OFF = TRUE THEN
				gServoHopperInterface.Commands.RequestMoveVelocity := FALSE;
				state := SERVOHOPPER_IDLE;
			ELSIF AtTorqueTimer.Q THEN
				gServoHopperInterface.Parameters.MovementParameters.Direction := 1;
				gServoHopperInterface.Commands.ToMapp.Update := TRUE;
				gServoHopperInterface.Commands.RequestMoveVelocity := TRUE;
				state := SERVOHOPPER_COOLDOWN;
			END_IF

		SERVOHOPPER_COOLDOWN:

			StartDwellTimer.IN := TRUE;

			IF gIO.DIs.HopperMotor_OFF = TRUE THEN
				gServoHopperInterface.Commands.RequestMoveVelocity := FALSE;
				state := SERVOHOPPER_IDLE;
			ELSIF StartDwellTimer.Q THEN
				gServoHopperInterface.Parameters.MovementParameters.Direction := 0;
				gServoHopperInterface.Commands.ToMapp.Update := TRUE;
				gServoHopperInterface.Commands.RequestMoveVelocity := TRUE;
				state := SERVOHOPPER_MOVE_VELOCITY;
			END_IF

		SERVOHOPPER_ERROR:

			gServoHopperInterface.Status.MoveComplete := TRUE;
			gHMI.Commands.StartServoHopper := FALSE;

			gServoHopperInterface.Commands.RequestMoveVelocity := FALSE;

			IF (gNumActiveAlarms = 0) THEN
				state := SERVOHOPPER_WAIT_FOR_HOME;
			END_IF

	END_CASE;

	StartDwellTimer.PT := gHMI.Parameters.ServoHopperDwellTime; //500 ms
	StartDwellTimer();

	AtTorqueTimer.PT := gHMI.Parameters.AtTorqueTime; //500 ms
	AtTorqueTimer();

END_PROGRAM

PROGRAM _EXIT
				(* Insert code here *)

END_PROGRAM
```

- Data object Logical/ServoMotion/acp10etxen (Ett) (no source held here)

### Program Logical/ServoMotion/MappCalls (IEC)

#### Cyclic.ld - Cyclic code
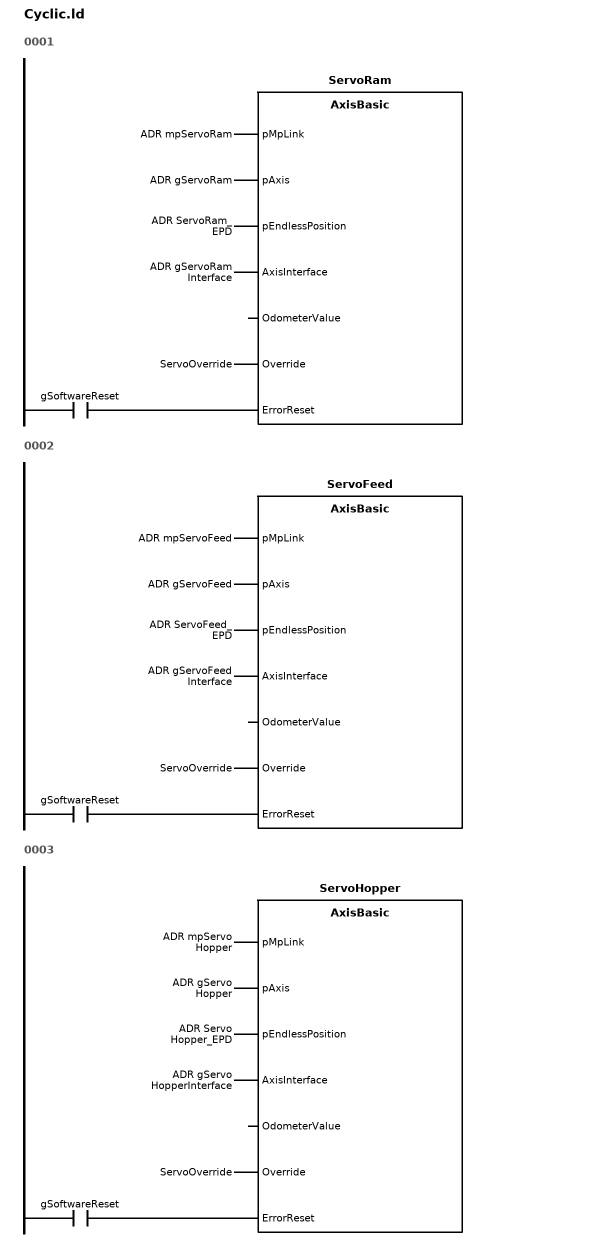
Ladder, written as Structured Text:
```iecst
PROGRAM _CYCLIC
(* Network 1 *)
ServoRam(pMpLink := ADR(mpServoRam), pAxis := ADR(gServoRam), pEndlessPosition := ADR(ServoRam_EPD), AxisInterface := ADR(gServoRamInterface), Override := ServoOverride, ErrorReset := gSoftwareReset);

(* Network 2 *)
ServoFeed(pMpLink := ADR(mpServoFeed), pAxis := ADR(gServoFeed), pEndlessPosition := ADR(ServoFeed_EPD), AxisInterface := ADR(gServoFeedInterface), Override := ServoOverride, ErrorReset := gSoftwareReset);

(* Network 3 *)
ServoHopper(pMpLink := ADR(mpServoHopper), pAxis := ADR(gServoHopper), pEndlessPosition := ADR(ServoHopper_EPD), AxisInterface := ADR(gServoHopperInterface), Override := ServoOverride, ErrorReset := gSoftwareReset);
END_PROGRAM
```

#### Init.st
```iecst
PROGRAM _INIT

	ServoOverride := 1.0;

END_PROGRAM
```

#### Variables.var - Local variables
```iecst
VAR
	ServoHopper : AxisBasic;
	ServoFeed : AxisBasic;
	ServoRam : AxisBasic;
	ServoOverride : REAL := 1.0;
END_VAR
```

### Program Logical/ServoMotion/MotionHandler (ANSIC)

#### Main.c - Init, cyclic, exit code
```c
#include <bur/plctypes.h>

#ifdef _DEFAULT_INCLUDES
#include <AsDefault.h>
#endif

/**
* This task:
*
* Populates homing and coupling defaults for each axis
* Instantiates axis control state machines for each axis
*
*
*/

void _INIT ProgramInit(void)
{

	gHomingParameters.ServoRam.Mode = mpAXIS_HOME_MODE_BLOCK_DS; //Servo Ram homes to hard stop
	gHomingParameters.ServoRam.BlockDetectionPositionError = 1.5;
	gHomingParameters.ServoRam.PositionErrorStopLimit = 2.0;
	gHomingParameters.ServoRam.StartDirection = mpAXIS_HOME_DIR_NEGATIVE;
	gHomingParameters.ServoRam.HomingDirection = mpAXIS_HOME_DIR_POSITIVE;
	gHomingParameters.ServoRam.StartVelocity = 10;
	gHomingParameters.ServoRam.HomingVelocity = 5;
	gHomingParameters.ServoRam.Position = -12.5;
	gHomingParameters.ServoRam.SensorOffset = 12.5; //back off switch by 12.5 mm and call that position home
	gHomingParameters.ServoRam.TorqueLimit = 2.0;

	gHomingParameters.ServoFeed.Mode = mpAXIS_HOME_MODE_DIRECT;
	gHomingParameters.ServoFeed.StartDirection = mpAXIS_HOME_DIR_NEGATIVE;
	gHomingParameters.ServoFeed.HomingDirection = mpAXIS_HOME_DIR_POSITIVE;
	gHomingParameters.ServoFeed.Position = 0;
	gHomingParameters.ServoFeed.SensorOffset = 0;

	gHomingParameters.ServoHopper.Mode = mpAXIS_HOME_MODE_DIRECT;
	gHomingParameters.ServoHopper.StartDirection = mpAXIS_HOME_DIR_NEGATIVE;
	gHomingParameters.ServoHopper.HomingDirection = mpAXIS_HOME_DIR_POSITIVE;
	gHomingParameters.ServoHopper.Position = 0;
	gHomingParameters.ServoHopper.SensorOffset = 0;

	ServoRamFirstHomeExecuted = 0; //THIS MUST ALWAYS BE SET TO FALSE. THIS IS A SINGLE TURN ENCODER
	ServoFeedFirstHomeExecuted = 0; //THIS MUST ALWAYS BE SET TO FALSE. THIS IS A SINGLE TURN ENCODER
	ServoHopperFirstHomeExecuted = 0; //THIS MUST ALWAYS BE SET TO FALSE. THIS IS A SINGLE TURN ENCODER

	//******* Start Axis and Drive Param Default Settings *******//

	//ram

	strcpy((char*)&gServoRamInterface.Parameters.AxisAndDrivePars.AxisName, "Ram");
	gServoRamInterface.Parameters.AxisAndDrivePars.Axis.BaseType = mpAXIS_LIMITED_LINEAR;
	gServoRamInterface.Parameters.AxisAndDrivePars.Axis.MeasurementUnit = mpAXIS_UNIT_MM;
	gServoRamInterface.Parameters.AxisAndDrivePars.Axis.MeasurementResolution = 0.01;
	gServoRamInterface.Parameters.AxisAndDrivePars.Axis.SoftwareLimitPositions.LowerLimit = 0;
	gServoRamInterface.Parameters.AxisAndDrivePars.Axis.SoftwareLimitPositions.UpperLimit = 550.0;
	gServoRamInterface.Parameters.AxisAndDrivePars.Axis.PeriodSettings.Period = 360;

	gServoRamInterface.Parameters.AxisAndDrivePars.Axis.MovementLimits.VelocityPositive = 1000.0;
	gServoRamInterface.Parameters.AxisAndDrivePars.Axis.MovementLimits.VelocityNegative = 1000.0;
	gServoRamInterface.Parameters.AxisAndDrivePars.Axis.MovementLimits.Acceleration = 5000.0;
	gServoRamInterface.Parameters.AxisAndDrivePars.Axis.MovementLimits.Deceleration = 5000.0;
	gServoRamInterface.Parameters.AxisAndDrivePars.Axis.MovementLimits.JerkTime = 0.0;
	gServoRamInterface.Parameters.AxisAndDrivePars.Axis.MovementLimits.PositionErrorStopLimit = 12;
	gServoRamInterface.Parameters.AxisAndDrivePars.Axis.MovementLimits.VelocityErrorStopLimit = 0.0;
	gServoRamInterface.Parameters.AxisAndDrivePars.Axis.MovementLimits.VelocityErrorStopLimitMode = mpAXIS_VEL_MODE_OFF;

	//gServoRamInterface.Parameters.AxisAndDrivePars.Axis.CyclicReadChannels.UserChannelParameterID = 214;

	gServoRamInterface.Parameters.AxisAndDrivePars.Drive.Gearbox.Input = 7;
	gServoRamInterface.Parameters.AxisAndDrivePars.Drive.Gearbox.Output = 1;
	gServoRamInterface.Parameters.AxisAndDrivePars.Drive.Gearbox.Direction = mpAXIS_DIR_CLOCKWISE;

	gServoRamInterface.Parameters.AxisAndDrivePars.Drive.Transformation.ReferenceDistance = 245.53333;

	//gServoRamInterface.Parameters.AxisAndDrivePars.Drive.Controller.Mode = mpAXIS_CTRL_MODE_POSITION_FF;
	gServoRamInterface.Parameters.AxisAndDrivePars.Drive.Controller.Mode = mpAXIS_CTRL_MODE_POSITION;
	gServoRamInterface.Parameters.AxisAndDrivePars.Drive.Controller.Position.ProportionalGain = 250.0;
	gServoRamInterface.Parameters.AxisAndDrivePars.Drive.Controller.Position.IntegralTime = 0.0;
	gServoRamInterface.Parameters.AxisAndDrivePars.Drive.Controller.Position.PredictionTime = 0.0004;
	gServoRamInterface.Parameters.AxisAndDrivePars.Drive.Controller.Position.TotalDelayTime = 0.0004;

	gServoRamInterface.Parameters.AxisAndDrivePars.Drive.Controller.Speed.ProportionalGain = 7.5;
	gServoRamInterface.Parameters.AxisAndDrivePars.Drive.Controller.Speed.IntegralTime = 0.1;
	gServoRamInterface.Parameters.AxisAndDrivePars.Drive.Controller.Speed.FilterTime = 0.0;

	//these values are only used if controller mode is set to position + feed forward
	gServoRamInterface.Parameters.AxisAndDrivePars.Drive.Controller.FeedForward.TorqueLoad = 0.0;
	gServoRamInterface.Parameters.AxisAndDrivePars.Drive.Controller.FeedForward.TorquePositive = 0.0;
	gServoRamInterface.Parameters.AxisAndDrivePars.Drive.Controller.FeedForward.TorqueNegative = 0.0;
	gServoRamInterface.Parameters.AxisAndDrivePars.Drive.Controller.FeedForward.SpeedTorqueFactor = 0.0;
	gServoRamInterface.Parameters.AxisAndDrivePars.Drive.Controller.FeedForward.Inertia = 0.0;
	gServoRamInterface.Parameters.AxisAndDrivePars.Drive.Controller.FeedForward.AccelerationFilterTime = 0.0;

	//feed

	strcpy((char*)&gServoFeedInterface.Parameters.AxisAndDrivePars.AxisName, "Feed");
	gServoFeedInterface.Parameters.AxisAndDrivePars.Axis.BaseType = mpAXIS_PERIODIC_ROTARY;
	gServoFeedInterface.Parameters.AxisAndDrivePars.Axis.MeasurementUnit = mpAXIS_UNIT_DEGREES;
	gServoFeedInterface.Parameters.AxisAndDrivePars.Axis.MeasurementResolution = 0.01;
	gServoFeedInterface.Parameters.AxisAndDrivePars.Axis.SoftwareLimitPositions.LowerLimit = 0;
	gServoFeedInterface.Parameters.AxisAndDrivePars.Axis.SoftwareLimitPositions.UpperLimit = 360.0;
	gServoFeedInterface.Parameters.AxisAndDrivePars.Axis.PeriodSettings.Period = 360.0;

	gServoFeedInterface.Parameters.AxisAndDrivePars.Axis.MovementLimits.VelocityPositive = 3600.0;
	gServoFeedInterface.Parameters.AxisAndDrivePars.Axis.MovementLimits.VelocityNegative = 3600.0;
	gServoFeedInterface.Parameters.AxisAndDrivePars.Axis.MovementLimits.Acceleration = 36000.0;
	gServoFeedInterface.Parameters.AxisAndDrivePars.Axis.MovementLimits.Deceleration = 36000.0;
	gServoFeedInterface.Parameters.AxisAndDrivePars.Axis.MovementLimits.JerkTime = 0.0;
	gServoFeedInterface.Parameters.AxisAndDrivePars.Axis.MovementLimits.PositionErrorStopLimit = 2;
	gServoFeedInterface.Parameters.AxisAndDrivePars.Axis.MovementLimits.VelocityErrorStopLimit = 0.0;
	gServoFeedInterface.Parameters.AxisAndDrivePars.Axis.MovementLimits.VelocityErrorStopLimitMode = mpAXIS_VEL_MODE_OFF;

	//gServoFeedInterface.Parameters.AxisAndDrivePars.Axis.CyclicReadChannels.UserChannelParameterID = 214;

	gServoFeedInterface.Parameters.AxisAndDrivePars.Drive.Gearbox.Input = 15;
	gServoFeedInterface.Parameters.AxisAndDrivePars.Drive.Gearbox.Output = 1;
	gServoFeedInterface.Parameters.AxisAndDrivePars.Drive.Gearbox.Direction = mpAXIS_DIR_COUNTERCLOCKWISE;

	gServoFeedInterface.Parameters.AxisAndDrivePars.Drive.Transformation.ReferenceDistance = 360.0;

	//gServoFeedInterface.Parameters.AxisAndDrivePars.Drive.Controller.Mode = mpAXIS_CTRL_MODE_POSITION_FF;
	gServoFeedInterface.Parameters.AxisAndDrivePars.Drive.Controller.Mode = mpAXIS_CTRL_MODE_POSITION;
	gServoFeedInterface.Parameters.AxisAndDrivePars.Drive.Controller.Position.ProportionalGain = 400.0;
	gServoFeedInterface.Parameters.AxisAndDrivePars.Drive.Controller.Position.IntegralTime = 0.0;
	gServoFeedInterface.Parameters.AxisAndDrivePars.Drive.Controller.Position.PredictionTime = 0.0004;
	gServoFeedInterface.Parameters.AxisAndDrivePars.Drive.Controller.Position.TotalDelayTime = 0.0004;

	gServoFeedInterface.Parameters.AxisAndDrivePars.Drive.Controller.Speed.ProportionalGain = 0.6;
	gServoFeedInterface.Parameters.AxisAndDrivePars.Drive.Controller.Speed.IntegralTime = 0.1;
	gServoFeedInterface.Parameters.AxisAndDrivePars.Drive.Controller.Speed.FilterTime = 0.0;

	//these values are only used if controller mode is set to position + feed forward
	gServoFeedInterface.Parameters.AxisAndDrivePars.Drive.Controller.FeedForward.TorqueLoad = 0.0;
	gServoFeedInterface.Parameters.AxisAndDrivePars.Drive.Controller.FeedForward.TorquePositive = 0.0;
	gServoFeedInterface.Parameters.AxisAndDrivePars.Drive.Controller.FeedForward.TorqueNegative = 0.0;
	gServoFeedInterface.Parameters.AxisAndDrivePars.Drive.Controller.FeedForward.SpeedTorqueFactor = 0.0;
	gServoFeedInterface.Parameters.AxisAndDrivePars.Drive.Controller.FeedForward.Inertia = 0.0;
	gServoFeedInterface.Parameters.AxisAndDrivePars.Drive.Controller.FeedForward.AccelerationFilterTime = 0.0;

	//hopper

	strcpy((char*)&gServoHopperInterface.Parameters.AxisAndDrivePars.AxisName, "Hopper");
	gServoHopperInterface.Parameters.AxisAndDrivePars.Axis.BaseType = mpAXIS_LINEAR;
	gServoHopperInterface.Parameters.AxisAndDrivePars.Axis.MeasurementUnit = mpAXIS_UNIT_MM;
	gServoHopperInterface.Parameters.AxisAndDrivePars.Axis.MeasurementResolution = 0.01;
	gServoHopperInterface.Parameters.AxisAndDrivePars.Axis.SoftwareLimitPositions.LowerLimit = 0;
	gServoHopperInterface.Parameters.AxisAndDrivePars.Axis.SoftwareLimitPositions.UpperLimit = 100.0;
	gServoHopperInterface.Parameters.AxisAndDrivePars.Axis.PeriodSettings.Period = 360;

	gServoHopperInterface.Parameters.AxisAndDrivePars.Axis.MovementLimits.VelocityPositive = 1000.0;
	gServoHopperInterface.Parameters.AxisAndDrivePars.Axis.MovementLimits.VelocityNegative = 1000.0;
	gServoHopperInterface.Parameters.AxisAndDrivePars.Axis.MovementLimits.Acceleration = 5000.0;
	gServoHopperInterface.Parameters.AxisAndDrivePars.Axis.MovementLimits.Deceleration = 5000.0;
	gServoHopperInterface.Parameters.AxisAndDrivePars.Axis.MovementLimits.JerkTime = 0.0;
	gServoHopperInterface.Parameters.AxisAndDrivePars.Axis.MovementLimits.PositionErrorStopLimit = 2;
	gServoHopperInterface.Parameters.AxisAndDrivePars.Axis.MovementLimits.VelocityErrorStopLimit = 0.0;
	gServoHopperInterface.Parameters.AxisAndDrivePars.Axis.MovementLimits.VelocityErrorStopLimitMode = mpAXIS_VEL_MODE_OFF;

	//gServoHopperInterface.Parameters.AxisAndDrivePars.Axis.CyclicReadChannels.UserChannelParameterID = 214;

	gServoHopperInterface.Parameters.AxisAndDrivePars.Drive.Gearbox.Input = 10;
	gServoHopperInterface.Parameters.AxisAndDrivePars.Drive.Gearbox.Output = 1;
	gServoHopperInterface.Parameters.AxisAndDrivePars.Drive.Gearbox.Direction = mpAXIS_DIR_CLOCKWISE;

	gServoHopperInterface.Parameters.AxisAndDrivePars.Drive.Transformation.ReferenceDistance = 127;

	//gServoHopperInterface.Parameters.AxisAndDrivePars.Drive.Controller.Mode = mpAXIS_CTRL_MODE_POSITION_FF;
	gServoHopperInterface.Parameters.AxisAndDrivePars.Drive.Controller.Mode = mpAXIS_CTRL_MODE_POSITION;
	gServoHopperInterface.Parameters.AxisAndDrivePars.Drive.Controller.Position.ProportionalGain = 400.0;
	gServoHopperInterface.Parameters.AxisAndDrivePars.Drive.Controller.Position.IntegralTime = 0.0;
	gServoHopperInterface.Parameters.AxisAndDrivePars.Drive.Controller.Position.PredictionTime = 0.0004;
	gServoHopperInterface.Parameters.AxisAndDrivePars.Drive.Controller.Position.TotalDelayTime = 0.0004;

	gServoHopperInterface.Parameters.AxisAndDrivePars.Drive.Controller.Speed.ProportionalGain = 0.6;
	gServoHopperInterface.Parameters.AxisAndDrivePars.Drive.Controller.Speed.IntegralTime = 0.1;
	gServoHopperInterface.Parameters.AxisAndDrivePars.Drive.Controller.Speed.FilterTime = 0.0;

	//these values are only used if controller mode is set to position + feed forward
	gServoHopperInterface.Parameters.AxisAndDrivePars.Drive.Controller.FeedForward.TorqueLoad = 0.0;
	gServoHopperInterface.Parameters.AxisAndDrivePars.Drive.Controller.FeedForward.TorquePositive = 0.0;
	gServoHopperInterface.Parameters.AxisAndDrivePars.Drive.Controller.FeedForward.TorqueNegative = 0.0;
	gServoHopperInterface.Parameters.AxisAndDrivePars.Drive.Controller.FeedForward.SpeedTorqueFactor = 0.0;
	gServoHopperInterface.Parameters.AxisAndDrivePars.Drive.Controller.FeedForward.Inertia = 0.0;
	gServoHopperInterface.Parameters.AxisAndDrivePars.Drive.Controller.FeedForward.AccelerationFilterTime = 0.0;

	//******* End Axis and Drive Param Default Settings *******//

}

void _CYCLIC ProgramCyclic(void)
{

	//******************START RAM HANDLER******************//
	gIsSimulated = DiagCpuIsSimulated();

	if (ServoRamFirstHomeExecuted == 0) {
		gHMI.StatusDatapoints.ServoRamHomeSDP = UNHIDE;
	} else {
		gHMI.StatusDatapoints.ServoRamHomeSDP = HIDE;
	}

	gServoRamInterface.Commands.RequestHome = gHMI.Commands.HomeServoRam || ServoRamAutoHome;
	gServoRamInterface.Commands.RequestJogPos = gHMI.Commands.JogServoRamPos;
	gServoRamInterface.Commands.RequestJogNeg = gHMI.Commands.JogServoRamNeg;
	gServoRamInterface.Parameters.MovementParameters.Jog.Acceleration = gHMI.Parameters.ServoRamAccel;
	gServoRamInterface.Parameters.MovementParameters.Jog.Deceleration = gHMI.Parameters.ServoRamAccel;
	gServoRamInterface.Parameters.MovementParameters.Jog.Velocity = gHMI.Parameters.ServoRamJogVelocity;

	gServoRamInterface.Parameters.MovementParameters.Acceleration = gHMI.Parameters.ServoRamAccel;
	gServoRamInterface.Parameters.MovementParameters.Deceleration = gHMI.Parameters.ServoRamAccel;
	gServoRamInterface.Parameters.MovementParameters.Torque.Limit = gHMI.Parameters.ServoRamTorqueLimit;
	gServoRamInterface.Parameters.MovementParameters.CyclicRead.TorqueMode = mpAXIS_READ_CYCLIC;

	//update torque limit anytime it is changed
	if (gServoRamInterface.Status.AxisInitialized) {
		if (OldTorqueLimitRam != gServoRamInterface.Parameters.MovementParameters.Torque.Limit) {
			gServoRamInterface.Commands.ToMapp.Update = 1;
		}

		OldTorqueLimitRam = gServoRamInterface.Parameters.MovementParameters.Torque.Limit;
	}

	//home request while running should clear command to cycle the ram This prevents ram from taking off immediately after home complets
	if (gServoRamInterface.Commands.RequestHome) {
		gHMI.Commands.CycleServoRam = 0;
	}

	//OldTorqueLimitRam = gServoRamInterface.Parameters.MovementParameters.Torque.Limit;

	ServoRamHandler.AlarmActive = gHighSeverityAlarmActive;
	ServoRamHandler.IsSimulated = gIsSimulated;
	ServoRamHandler.FirstHomeExecuted = &ServoRamFirstHomeExecuted;
	ServoRamHandler.pInterface = &gServoRamInterface;
	ServoRamHandler.pHomingParameters = &gHomingParameters.ServoRam;
	AxisHandler(&ServoRamHandler);
	//******************END RAM HANDLER******************//

	//******************START FEED HANDLER******************//
	gServoFeedInterface.Commands.RequestHome = gHMI.Commands.HomeServoFeed;
	gServoFeedInterface.Commands.RequestJogPos = gHMI.Commands.JogServoFeedPos;
	gServoFeedInterface.Commands.RequestJogNeg = gHMI.Commands.JogServoFeedNeg;
	gServoFeedInterface.Parameters.MovementParameters.Jog.Acceleration = gHMI.Parameters.ServoFeedAccel;
	gServoFeedInterface.Parameters.MovementParameters.Jog.Deceleration = gHMI.Parameters.ServoFeedAccel;
	gServoFeedInterface.Parameters.MovementParameters.Jog.Velocity = gHMI.Parameters.ServoFeedJogVelocity;

	gServoFeedInterface.Parameters.MovementParameters.Acceleration = gHMI.Parameters.ServoFeedAccel;
	gServoFeedInterface.Parameters.MovementParameters.Deceleration = gHMI.Parameters.ServoFeedAccel;
	gServoFeedInterface.Parameters.MovementParameters.Velocity = gHMI.Parameters.ServoFeedVelocity;
	gServoFeedInterface.Parameters.MovementParameters.Torque.Limit = gHMI.Parameters.ServoFeedTorqueLimit;

	//update torque limit anytime it is changed
	if (gServoFeedInterface.Status.AxisInitialized) {
		if (OldTorqueLimitFeed != gServoFeedInterface.Parameters.MovementParameters.Torque.Limit) {
			gServoFeedInterface.Commands.ToMapp.Update = 1;
		}

		OldTorqueLimitFeed = gServoFeedInterface.Parameters.MovementParameters.Torque.Limit;
	}

	ServoFeedHandler.AlarmActive = gHighSeverityAlarmActive;
	ServoFeedHandler.IsSimulated = gIsSimulated;
	ServoFeedHandler.FirstHomeExecuted = &ServoFeedFirstHomeExecuted;
	ServoFeedHandler.pInterface = &gServoFeedInterface;
	ServoFeedHandler.pHomingParameters = &gHomingParameters.ServoFeed;
	AxisHandler(&ServoFeedHandler);
	//******************END FEED HANDLER******************//

	//******************START FEED HANDLER******************//
	gServoHopperInterface.Commands.RequestHome = gHMI.Commands.HomeServoHopper;
	gServoHopperInterface.Commands.RequestJogPos = gHMI.Commands.JogServoHopperPos;
	gServoHopperInterface.Commands.RequestJogNeg = gHMI.Commands.JogServoHopperNeg;
	gServoHopperInterface.Parameters.MovementParameters.Jog.Acceleration = gHMI.Parameters.ServoHopperAccel;
	gServoHopperInterface.Parameters.MovementParameters.Jog.Deceleration = gHMI.Parameters.ServoHopperAccel;
	gServoHopperInterface.Parameters.MovementParameters.Jog.Velocity = gHMI.Parameters.ServoHopperJogVelocity;

	gServoHopperInterface.Parameters.MovementParameters.Acceleration = gHMI.Parameters.ServoHopperAccel;
	gServoHopperInterface.Parameters.MovementParameters.Deceleration = gHMI.Parameters.ServoHopperAccel;
	gServoHopperInterface.Parameters.MovementParameters.Velocity = gHMI.Parameters.ServoHopperVelocity;
	gServoHopperInterface.Parameters.MovementParameters.Torque.Limit = gHMI.Parameters.ServoHopperTorqueLimit;
	gServoHopperInterface.Parameters.MovementParameters.CyclicRead.TorqueMode = mpAXIS_READ_CYCLIC;

	//update torque limit anytime it is changed
	if (gServoHopperInterface.Status.AxisInitialized) {
		if (OldTorqueLimitHopper != gServoHopperInterface.Parameters.MovementParameters.Torque.Limit) {
			gServoHopperInterface.Commands.ToMapp.Update = 1;
		}

		OldTorqueLimitHopper = gServoHopperInterface.Parameters.MovementParameters.Torque.Limit;
	}

	ServoHopperHandler.AlarmActive = gHighSeverityAlarmActive;
	ServoHopperHandler.IsSimulated = gIsSimulated;
	ServoHopperHandler.FirstHomeExecuted = &ServoHopperFirstHomeExecuted;
	ServoHopperHandler.pInterface = &gServoHopperInterface;
	ServoHopperHandler.pHomingParameters = &gHomingParameters.ServoHopper;
	AxisHandler(&ServoHopperHandler);
	//******************END FEED HANDLER******************//

}

void _EXIT ProgramExit(void)
{

}
```

#### Variables.var - Local variables
```iecst
VAR
	ServoFeedHandler : AxisHandler;
	ServoHopperHandler : AxisHandler;
	ServoRamHandler : AxisHandler;
	OldTorqueLimitHopper : REAL;
	OldTorqueLimitFeed : REAL;
	OldTorqueLimitRam : REAL;
END_VAR
```

- NUMATICS-580-20150428-145500.xdd (not shown)

### Package Logical/gFeedobj - gFeedobj

### Data object Logical/gFeedobj/gHopa (Apt)

#### gHopa.apt
```
AcoposParameterTable:
  Root Parameters:
    230 = PCTRL_S_SET (Name=PCTRL_S_ACT_PARID)  // CTRL Position controller: Actual encoder position parameter ID
```

### Data object Logical/gFeedobj/gFeedi (Ax)

#### gFeedi.ax
```
InitParameter (Version=5.8.2, NcSwId=ACP10)
  ACP10AXIS_typ:
    dig_in:
      level:
        reference = ncACTIV_HI
        pos_hw_end = ncACTIV_HI
        neg_hw_end = ncACTIV_HI
        trigger1 = ncACTIV_HI
        trigger2 = ncACTIV_HI
    encoder_if:
      parameter:
        count_dir = ncSTANDARD
        scaling:
          load:
            units = 12700
            rev_motor = 10
    limit:
      parameter:
        v_pos = 100000.0
        v_neg = 100000.0
        a1_pos = 500000.0
        a2_pos = 500000.0
        a1_neg = 500000.0
        a2_neg = 500000.0
        t_jolt = 0.0
        t_in_pos = 0.0
        pos_sw_end = 10000
        neg_sw_end = 0
        ds_warning = 200.0
        ds_stop = 200.0
        a_stop = 1.0E+30
        dv_stop = 0.0
        dv_stop_mode = ncOFF
    controller:
      mode = ncPOSITION
      position:
        kv = 400.0
        tn = 0.0
        t_predict = 0.0004
        t_total = 0.0004
        p_max = 1.0E+30
        i_max = 1.0E+30
      speed:
        kv = 0.6
        tn = 0.1
        t_filter = 0.0
        isq_filter1:
          type = ncOFF
          a0 = 0.0
          a1 = 0.0
          b0 = 0.0
          b1 = 0.0
          b2 = 0.0
          c0_par_id = 0
          c1_par_id = 0
        isq_filter2:
          type = ncOFF
          a0 = 0.0
          a1 = 0.0
          b0 = 0.0
          b1 = 0.0
          b2 = 0.0
          c0_par_id = 0
          c1_par_id = 0
        isq_filter3:
          type = ncOFF
          a0 = 0.0
          a1 = 0.0
          b0 = 0.0
          b1 = 0.0
          b2 = 0.0
          c0_par_id = 0
          c1_par_id = 0
      uf:
        type = ncLINEAR
        auto_config = ncOFF
        u0 = 0.0
        un = 0.0
        fn = 0.0
        k_f_slip = 0.0
      ff:
        mode = ncSTANDARD
        torque_load = 0.0
        torque_pos = 0.0
        torque_neg = 0.0
        kv_torque = 0.0
        inertia = 0.0
        t_filter_a = 0.0
      fb:
        mode = ncSTANDARD
        speed_mix_ratio = 0.0
        speed_kv = 2.0
      model:
        mass1:
          inertia = 0.0
          viscous_friction = 0.0
        mass2:
          inertia = 0.0
          viscous_friction = 0.0
          stiffness = 0.0
          damping = 0.0
    move:
      stop:
        parameter[0]:
          decel_ramp = ncA_LIMIT
          controller = ncON
        parameter[1]:
          decel_ramp = ncA_LIMIT
          controller = ncON
        parameter[2]:
          decel_ramp = ncA_LIMIT
          controller = ncON
        parameter[3]:
          decel_ramp = ncA_LIMIT
          controller = ncON
        quickstop:
          decel_ramp = ncA_LIMIT
          t_jolt = 0.0
        drive_error:
          decel_ramp = ncA_LIMIT
      homing:
        parameter:
          s = 0
          v_switch = 5000.0
          v_trigger = 500.0
          a = 50000.0
          mode = ncDIRECT
          edge_sw = ncPOSITIVE
          start_dir = ncPOSITIVE
          trigg_dir = ncPOSITIVE
          ref_pulse = ncOFF
          fix_dir = ncOFF
          tr_s_block = 0.0
          torque_lim = 0.0
          ds_block = 0.0
          ds_stop = 0.0
      basis:
        parameter:
          v_pos = 635.0
          v_neg = 635.0
          a1_pos = 36000.0
          a2_pos = 36000.0
          a1_neg = 36000.0
          a2_neg = 36000.0
    message:
      text:
        parameter:
          format = ncBREAK
          columns = 80
          data_modul = acp10etxen
```

### Program Logical/Program (IEC)

#### Main.st
```iecst
PROGRAM _INIT
	(* Insert code here *)
	b_ModuleStatus;
	mb_Station 			:= 'IF2.ST1';
	Melter;
END_PROGRAM

PROGRAM _CYCLIC
	(* Insert code here *)
	FB_NDSN_MB_PBFlex_Ctrl(IN_b_Enable :=NOT  Melter.b_r_LostCommunication,
		IN_mb_station := mb_Station,
		Melter := Melter);
	FB_NDSN_MB_PBFlex_Proc(IN_b_Enable :=NOT  Melter.b_r_LostCommunication,
		IN_mb_station := mb_Station,
		Melter := Melter);
	Melter.b_r_LostCommunication := NOT b_ModuleStatus;

END_PROGRAM

PROGRAM _EXIT
	(* Insert code here *)

END_PROGRAM
```

Listed in the project but not available here: Logical/Global.typ, Logical/Libraries/Vacuum/Types.typ, Logical/Libraries/Vacuum/Constants.var, Logical/Libraries/FoldPush/Types.typ, Logical/Libraries/FoldPush/Constants.var, Logical/Libraries/SetRamPars/Types.typ, Logical/Libraries/SetRamPars/Constants.var, Logical/Libraries/GrayToBin/Types.typ, Logical/Libraries/GrayToBin/Constants.var, Logical/Libraries/DistCalc/Types.typ, Logical/Libraries/DistCalc/Constants.var, Logical/Libraries/MappCall/Types.typ, Logical/Libraries/AxisFUBs/Types.typ, Logical/Libraries/AxisFUBs/Constants.var, Logical/Libraries/Lib_PBFlx/Constants.var, Logical/ModeControl/ModeControl/LocalFunctions.fun, Logical/ModeControl/ModeControl_ST/LocalFunctions.fun, Logical/Actuators/FoldPushControl/Init.ld, Logical/Actuators/FoldPushControl/Types.typ, Logical/Actuators/VacuumControl/Types.typ, Logical/AlarmControl/AlarmHandling/Types.typ, Logical/ncsdcctrl/ncsdcctrl.typ, Logical/ncsdcctrl/ncsdcctrl.var, Logical/gAxis01obj, Logical/EncoderDecoding/Init.c, Logical/EncoderDecoding/Exit.c, Logical/EncoderDecoding/Types.typ, Logical/ServoMotion/MappCalls/Exit.ld, Logical/ServoMotion/MappCalls/Types.typ, Logical/ServoMotion/MotionHandler/Types.typ
